// TIA Portal V21 export
FUNCTION_BLOCK "FB318"   // FB318, LAD
TITLE = FB318
{ S7_Optimized_Access := 'FALSE' }
AUTHOR : PRECISE
FAMILY : PRECISE
// VALVE TOGGLE
// stored: AutoNumber false, SetENOAutomatically false
   VAR_INPUT
      Enable : Bool;
      Disable : Bool;
      Fault : Bool;
      SecPulse : Bool;
      AlwaysTrue : Bool;
      StartConfirmationPopupSel : Bool;   // StartConfirmationPopupSel: 0-NO/1-YES
      EndConfirmationPopupSel : Bool;   // EndConfirmationPopupSel: 0-NO/1-YES
   END_VAR
   VAR_OUTPUT
      Valve : Bool;
      StartConfirmationPopup : Bool;   // For Start Confirmation Popup Selection: Yes
      EndConfirmationPopup : Bool;   // For End Confirmation Popup Selection: Yes
      PrintTrigger : Bool;
      PrintWord : Int;
      PrintStatus : String[50];
   END_VAR
   VAR_IN_OUT
      Open : Bool;
      Close : Bool;
      StartConfirmationAck : Bool;   // For Start Confirmation Popup Selection: Yes
      EndConfirmationAck : Bool;   // For End Confirmation Popup Selection: Yes
      SpareBtn1 : Bool;
      SpareBtn2 : Bool;
      SpareBtn3 : Bool;
      SpareBtn4 : Bool;
      Running : Bool;
      Selected : Bool;
      Over : Bool;
      StartConfirmationPopupTemp : Bool;   // For Start Confirmation Popup Selection: Yes
      EndConfirmationPopupTemp : Bool;   // For End Confirmation Popup Selection: Yes
   END_VAR
   VAR
      PrintTriggerTemp : Bool;
      RE1 : Bool;
      RE2 : Bool;
      RE3 : Bool;
      RE4 : Bool;
      RE5 : Bool;
      RE6 : Bool;
      RE7 : Bool;
      PrintTriggerResetTimer { S7_SetPoint := 'True'} : TON_TIME;
      BtnResetTimer { S7_SetPoint := 'True'} : TON_TIME;
   END_VAR
   VAR_TEMP   // added for the SCL form of the ladder/FBD networks
      _w1 : Bool;
      _w2 : Bool;
   END_VAR
BEGIN

REGION Network 1: Running
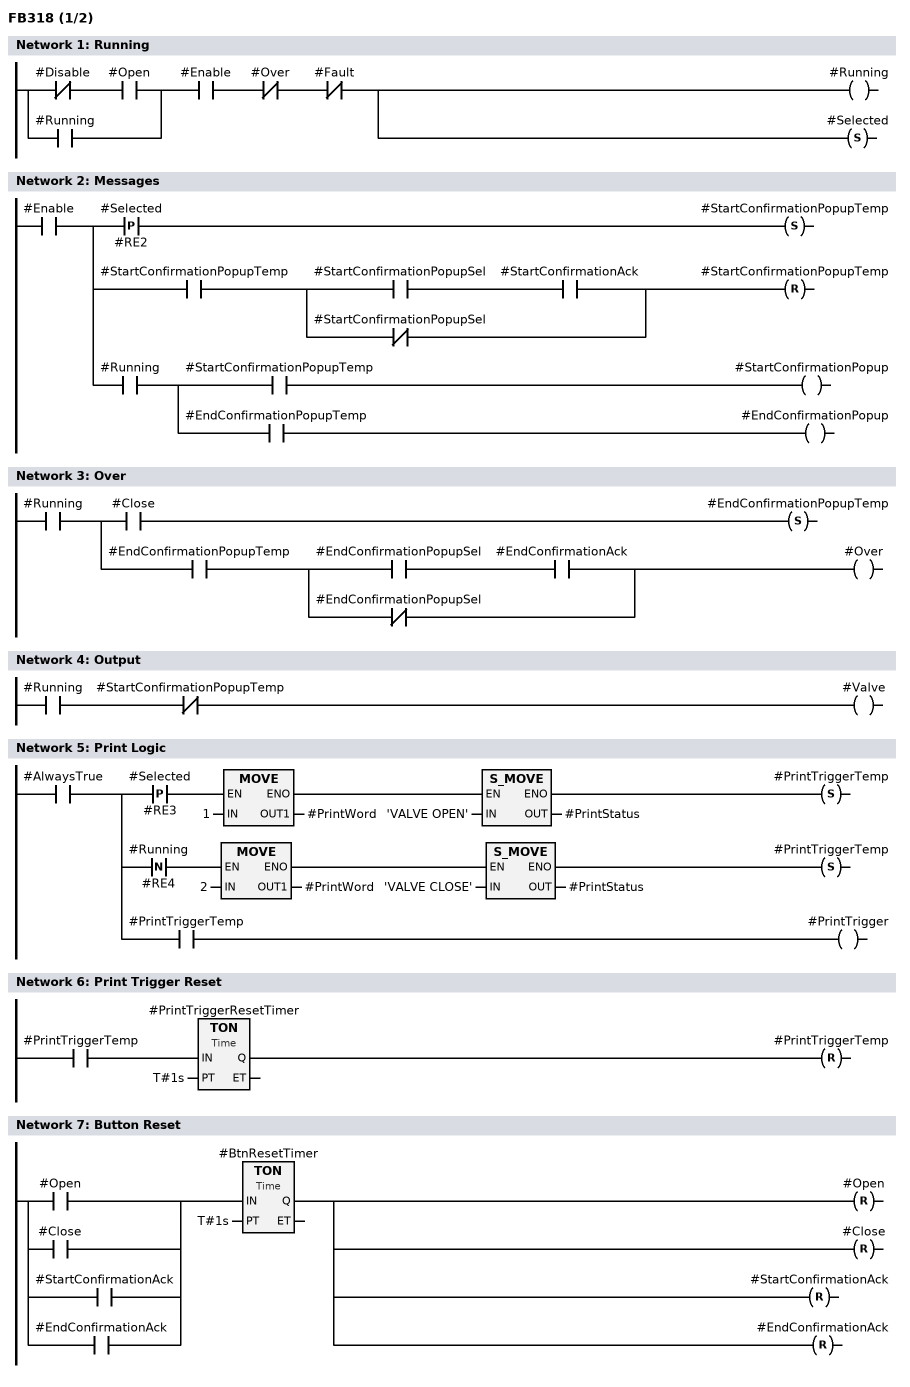
   RUNG wire#powerrail
      I_Contact( #Disable )
      Contact( #Open )
      wire#w1
      Contact( #Enable )
      I_Contact( #Over )
      I_Contact( #Fault )
      wire#w2
      Coil( #Running )
   END_RUNG
   RUNG wire#powerrail
      Contact( #Running )
   END_RUNG wire#w1
   RUNG wire#w2
      S_Coil( #Selected )
   END_RUNG
   // the same network as SCL:
   #Running := ((NOT #Disable AND #Open) OR #Running) AND #Enable AND NOT #Over AND NOT #Fault;
   IF #Running THEN #Selected := TRUE; END_IF;
END_REGION

REGION Network 2: Messages
   RUNG wire#powerrail
      Contact( #Enable )
      wire#w1
      P_Contact(operand := #Selected, bit := #RE2)
      S_Coil( #StartConfirmationPopupTemp )
   END_RUNG
   RUNG wire#w1
      Contact( #StartConfirmationPopupTemp )
      wire#w2
      Contact( #StartConfirmationPopupSel )
      Contact( #StartConfirmationAck )
      wire#w3
      R_Coil( #StartConfirmationPopupTemp )
   END_RUNG
   RUNG wire#w2
      I_Contact( #StartConfirmationPopupSel )
   END_RUNG wire#w3
   RUNG wire#w1
      Contact( #Running )
      wire#w4
      Contact( #StartConfirmationPopupTemp )
      Coil( #StartConfirmationPopup )
   END_RUNG
   RUNG wire#w4
      Contact( #EndConfirmationPopupTemp )
      Coil( #EndConfirmationPopup )
   END_RUNG
   // the same network as SCL:
   #_w1 := #Enable AND #Selected AND NOT #RE2;   // rising edge of #Selected
   #RE2 := #Selected;
   IF #_w1 THEN #StartConfirmationPopupTemp := TRUE; END_IF;
   IF #Enable AND #StartConfirmationPopupTemp AND ((#StartConfirmationPopupSel AND #StartConfirmationAck) OR NOT #StartConfirmationPopupSel) THEN
       #StartConfirmationPopupTemp := FALSE;
   END_IF;
   #_w2 := #Enable AND #Running;
   #StartConfirmationPopup := #_w2 AND #StartConfirmationPopupTemp;
   #EndConfirmationPopup := #_w2 AND #EndConfirmationPopupTemp;
END_REGION

REGION Network 3: Over
   RUNG wire#powerrail
      Contact( #Running )
      wire#w1
      Contact( #Close )
      S_Coil( #EndConfirmationPopupTemp )
   END_RUNG
   RUNG wire#w1
      Contact( #EndConfirmationPopupTemp )
      wire#w2
      Contact( #EndConfirmationPopupSel )
      Contact( #EndConfirmationAck )
      wire#w3
      Coil( #Over )
   END_RUNG
   RUNG wire#w2
      I_Contact( #EndConfirmationPopupSel )
   END_RUNG wire#w3
   // the same network as SCL:
   IF #Running AND #Close THEN #EndConfirmationPopupTemp := TRUE; END_IF;
   #Over := #Running AND #EndConfirmationPopupTemp AND ((#EndConfirmationPopupSel AND #EndConfirmationAck) OR NOT #EndConfirmationPopupSel);
END_REGION

REGION Network 4: Output
   RUNG wire#powerrail
      Contact( #Running )
      I_Contact( #StartConfirmationPopupTemp )
      Coil( #Valve )
   END_RUNG
   // the same network as SCL:
   #Valve := #Running AND NOT #StartConfirmationPopupTemp;
END_REGION

REGION Network 5: Print Logic
   RUNG wire#powerrail
      Contact( #AlwaysTrue )
      wire#w1
      P_Contact(operand := #Selected, bit := #RE3)
      { S7_GenerateENO := "TRUE" } Move(in := 1, out1 => #PrintWord)
      S_Move(in := 'VALVE OPEN', out => #PrintStatus)
      S_Coil( #PrintTriggerTemp )
   END_RUNG
   RUNG wire#w1
      N_Contact(operand := #Running, bit := #RE4)
      { S7_GenerateENO := "TRUE" } Move(in := 2, out1 => #PrintWord)
      S_Move(in := 'VALVE CLOSE', out => #PrintStatus)
      S_Coil( #PrintTriggerTemp )
   END_RUNG
   RUNG wire#w1
      Contact( #PrintTriggerTemp )
      Coil( #PrintTrigger )
   END_RUNG
   // the same network as SCL:
   // ENO of a box is taken as its EN; it also drops when the box reports an error
   #_w1 := #AlwaysTrue AND #Selected AND NOT #RE3;   // rising edge of #Selected
   #RE3 := #Selected;
   IF #_w1 THEN
       #PrintWord := 1;
       #PrintStatus := 'VALVE OPEN';
       #PrintTriggerTemp := TRUE;
   END_IF;
   #_w2 := #AlwaysTrue AND NOT #Running AND #RE4;   // falling edge of #Running
   #RE4 := #Running;
   IF #_w2 THEN
       #PrintWord := 2;
       #PrintStatus := 'VALVE CLOSE';
       #PrintTriggerTemp := TRUE;
   END_IF;
   #PrintTrigger := #AlwaysTrue AND #PrintTriggerTemp;
END_REGION

REGION Network 6: Print Trigger Reset
   RUNG wire#powerrail
      Contact( #PrintTriggerTemp )
      { S7_Templates := "time_type := Time" } #PrintTriggerResetTimer.TON(pt := T#1s, et =>)
      R_Coil( #PrintTriggerTemp )
   END_RUNG
   // the same network as SCL:
   #PrintTriggerResetTimer(IN := #PrintTriggerTemp, PT := T#1s);   // TON
   IF #PrintTriggerResetTimer.Q THEN #PrintTriggerTemp := FALSE; END_IF;
END_REGION

REGION Network 7: Button Reset
   RUNG wire#powerrail
      Contact( #Open )
      wire#w1
      { S7_Templates := "time_type := Time" } #BtnResetTimer.TON(pt := T#1s, et =>)
      wire#w2
      R_Coil( #Open )
   END_RUNG
   RUNG wire#powerrail
      Contact( #Close )
   END_RUNG wire#w1
   RUNG wire#powerrail
      Contact( #StartConfirmationAck )
   END_RUNG wire#w1
   RUNG wire#powerrail
      Contact( #EndConfirmationAck )
   END_RUNG wire#w1
   RUNG wire#w2
      R_Coil( #Close )
   END_RUNG
   RUNG wire#w2
      R_Coil( #StartConfirmationAck )
   END_RUNG
   RUNG wire#w2
      R_Coil( #EndConfirmationAck )
   END_RUNG
   // the same network as SCL:
   #BtnResetTimer(IN := #Open OR #Close OR #StartConfirmationAck OR #EndConfirmationAck, PT := T#1s);   // TON
   IF #BtnResetTimer.Q THEN
       #Open := FALSE;
       #Close := FALSE;
       #StartConfirmationAck := FALSE;
       #EndConfirmationAck := FALSE;
   END_IF;
END_REGION

REGION Network 8: Reset
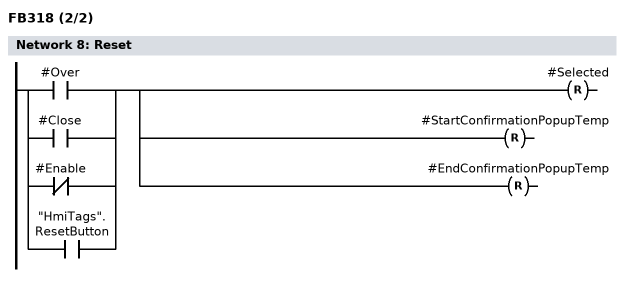
   RUNG wire#powerrail
      Contact( #Over )
      wire#w1
      R_Coil( #Selected )
   END_RUNG
   RUNG wire#powerrail
      Contact( #Close )
   END_RUNG wire#w1
   RUNG wire#powerrail
      I_Contact( #Enable )
   END_RUNG wire#w1
   RUNG wire#powerrail
      Contact( "HmiTags".ResetButton )
   END_RUNG wire#w1
   RUNG wire#w1
      R_Coil( #StartConfirmationPopupTemp )
   END_RUNG
   RUNG wire#w1
      R_Coil( #EndConfirmationPopupTemp )
   END_RUNG
   // the same network as SCL:
   IF #Over OR #Close OR NOT #Enable OR "HmiTags".ResetButton THEN
       #Selected := FALSE;
       #StartConfirmationPopupTemp := FALSE;
       #EndConfirmationPopupTemp := FALSE;
   END_IF;
END_REGION
END_FUNCTION_BLOCK
